FUNCTION_BLOCK FB_EventHTTP_Post
VAR_INPUT
	bSend		: BOOL;
	API_URI		: STRING[255];
	API_Msg		: STRING[255];
END_VAR
VAR_IN_OUT
	fbClient			: FB_IotHttpClient;
END_VAR
VAR_OUTPUT
	bSuccess			: Bool;
	bBusy				: BOOL;
	bError				: BOOL;
END_VAR
VAR	
	// set content to json
	API_STR     		: STRING(Tc3_IotBase.ParameterList.cSizeOfHttpContentType-1) := 'application/json';

	fbRequest			: FB_IotHttpRequest;
	fbHeader			: FB_IotHttpHeaderFieldMap;
	fbJson				: FB_JsonDomParser;
	
 	dtTimestamp    		: DATE_AND_TIME := DT#2017-04-04-12:42:42;
	fbJsonWriter		: FB_JsonDomParser;
	nState				: UDINT;
	RisingEdge			: R_TRIG;
	
	bGetContentResult	: BOOL;
	sContent			: STRING[5000] := ''; 
	
	bGetJsonResult		: BOOL;
	jsonDoc				: SJsonValue;
	jsonVal				: SJsonValue;
	sResultValue		: STRING;
	sResultValue2		: STRING;
	bOnce				: BOOL := TRUE;
	
	nReqCount			: UDINT;
	nResCount			: UDINT;
	nValidResCount		: UDINT;
	nErrCount			: UDINT;	
END_VAR

RisingEdge(CLK:= bSend);
IF bOnce THEN
	fbHeader.AddField('x-api-key', '8e0697a446bd2c17b4e1188f1d21439ef863aa79b59e31981a7135b3171f9b85', FALSE);	
	bOnce:= FALSE;
END_IF
CASE nState OF
0:		
	IF RisingEdge.Q THEN 
		sContent := API_Msg;
		fbRequest.sContentType := API_STR;
		IF fbRequest.SendRequest(sUri:= API_URI, fbClient:= fbClient, eRequestType:= ETcIotHttpRequestType.HTTP_POST, pContent:= ADR(sContent), nContentSize:= LEN2(ADR(sContent)), fbHeader) THEN				
			nState:= 1;
			bBusy:= TRUE;
			bError:= FALSE;
			bSuccess := FALSE;
		END_IF					
	END_IF
1:
	IF NOT fbRequest.bBusy THEN
		bError:= TRUE;
		IF NOT fbRequest.bError THEN
							 				
			bGetContentResult:= fbRequest.GetContent(pContent:= ADR(sContent), nContentSize:= SIZEOF(SContent), bSetNullTermination:= TRUE);	
			IF fbRequest.nStatusCode >= 200 AND fbRequest.nStatusCode < 300 THEN
				bGetJsonResult:= FALSE;
//				jsonDoc:= fbRequest.GetJsonDomContent(fbJson);				
//				IF jsonDoc <> 0 THEN
//					bGetJsonResult:= TRUE;
//					IF fbJson.HasMember(jsonDoc, 'status')  THEN
//						jsonVal:= fbJson.FindMember(jsonDoc, 'status');	
//						sResultValue:= fbJson.GetString(jsonVal);
//						IF sResultValue = 'success' THEN
							nValidResCount:= nValidResCount+1;	
							bSuccess := TRUE;
							bError:= FALSE;
//						END_IF
//					END_IF		
//				END_IF
				nResCount:= nResCount+1;					
			END_IF				
		END_IF
		nState:= 0;
		bBusy:= FALSE;
		IF bError THEN
			nErrCount:= nErrCount+1;
		END_IF		
	END_IF 
END_CASE

END_FUNCTION_BLOCK

(* stored: Version 1.1.0.1, ProductVersion 3.1.4024.12
   POU FB_EventHTTP_Post: Id {7187df70-8a1b-4d51-b4d1-62ad62dac9c6}, SpecialFunc None *)
